Staubli VAL3: JointFbkMsg.pjx

Parameters version=s7.7.2 stackSize=5000 millimeterUnit=true
Program file=start.pgx
Program file=stop.pgx
Data file=JointFbkMsg.dtx
Type name=Body path=Disk://Body/Body.pjx
Type name=Header path=Disk://Header/Header.pjx
Type name=Prefix path=Disk://Prefix/Prefix.pjx
Type name=JointFeedback path=Disk://JointFeedback/JointFeedback.pjx
